PROGRAM HMIUpdates
VAR
END_VAR

END_PROGRAM

(* stored: Version 1.1.0.1
   POU HMIUpdates: Id {27ceecba-ff72-431a-a52a-fe07066876e8}, SpecialFunc None *)
